Universal Robots URScript: 00B_05_Che_JIeXian.script

def P00B_05_Che_JIeXian():
  set_standard_analog_input_domain(0, 1)
  set_standard_analog_input_domain(1, 1)
  set_tool_analog_input_domain(0, 1)
  set_tool_analog_input_domain(1, 1)
  set_analog_outputdomain(0, 0)
  set_analog_outputdomain(1, 0)
  set_tool_voltage(0)
  set_input_actions_to_default()
  set_tcp(p[-0.06448999999999999,0.0207,0.28314999999999996,0.0,0.0,1.5902])
  set_payload(8.0)
  set_safety_mode_transition_hardness(1)
  set_gravity([0.0, 0.0, 9.82])
  $ 1 "机器人程序"
  $ 2 "MoveJ"
  $ 3 "路点_1"
  set_tcp(p[-0.06448999999999999,0.0207,0.28314999999999996,0.0,0.0,1.5902])
  movej(get_inverse_kin(p[.827586488288, -.301155839413, .786661241235, -.102992074225, .077805615287, -1.659522054939], qnear=[-0.16117841402162725, -1.8165248076068323, -1.8520506064044397, -1.153802220021383, -1.6081426779376429, 1.616330862045288]), a=0.6981317007977318, v=0.5235987755982988)
  $ 4 "路点_2"
  set_tcp(p[-0.06448999999999999,0.0207,0.28314999999999996,0.0,0.0,1.5902])
  movej(get_inverse_kin(p[.434262102635, .698472218287, .586851819079, -.148386171909, -.158137194586, -1.506962500167], qnear=[1.2591005563735962, -2.003486935292379, -2.0370481649981897, -0.8543809095965784, -1.6501196066485804, 0.34251177310943604]), a=0.6981317007977318, v=0.5235987755982988)
end
